Staubli VAL3: printArray.pgx

program printArray(string x_sFormat (dimensions=1), num& x_nArray[] (dimensions=1))
  local num i
begin
  for i=0 to size(x_nArray)-2
    put(toString(x_sFormat,x_nArray[i]))
    put(" ")
  endFor
  putln(toString(x_sFormat,x_nArray[size(x_nArray)-1]))
end
